// TIA Portal V18 export
DATA_BLOCK "ST10_DeviceError"   // DB1067
{ S7_Optimized_Access := 'FALSE' }
VERSION : 0.1
// stored: AutoNumber false, DBAccessibleFromOPCUA true, DBAccessibleFromWebserver true, IsOnlyStoredInLoadMemory false, IsWriteProtectedInAS false
   VAR RETAIN
      CylinderFault : Struct   // Cylinder Error（气缸错误）
         C1GoWorkFault : Bool;   // Cyl1
         C1GoHomeFault : Bool;   // Cyl1
         C1SensorPositionFault : Bool;   // Cyl1
         C1SpareFault : Bool;
         C2GoWorkFault : Bool;   // Cyl2
         C2GoHomeFault : Bool;   // Cyl2
         C2SensorPositionFault : Bool;   // Cyl2
         C2SpareFault : Bool;
         C3GoWorkFault : Bool;   // Cyl3
         C3GoHomeFault : Bool;   // Cyl3
         C3SensorPositionFault : Bool;   // Cyl3
         C3SpareFault : Bool;
         C4GoWorkFault : Bool;   // Cyl4
         C4GoHomeFault : Bool;   // Cyl4
         C4SensorPositionFault : Bool;   // Cyl4
         C4SpareFault : Bool;
         C5GoWorkFault : Bool;   // Cyl5
         C5GoHomeFault : Bool;   // Cyl5
         C5SensorPositionFault : Bool;   // Cyl5
         C5SpareFault : Bool;
         C6GoWorkFault : Bool;   // Cyl6
         C6GoHomeFault : Bool;   // Cyl6
         C6SensorPositionFault : Bool;   // Cyl6
         C6SpareFault : Bool;
         C7GoWorkFault : Bool;   // Cyl7
         C7GoHomeFault : Bool;   // Cyl7
         C7SensorPositionFault : Bool;   // Cyl7
         C7SpareFault : Bool;
         C8GoWorkFault : Bool;   // Cyl8
         C8GoHomeFault : Bool;   // Cyl8
         C8SensorPositionFault : Bool;   // Cyl8
         C8SpareFault : Bool;
         C9GoWorkFault : Bool;   // Cyl9
         C9GoHomeFault : Bool;   // Cyl9
         C9SensorPositionFault : Bool;   // Cyl9
         C9SpareFault : Bool;
         C10GoWorkFault : Bool;   // Cyl10
         C10GoHomeFault : Bool;   // Cyl10
         C10SensorPositionFault : Bool;   // Cyl10
         C10SpareFault : Bool;
         C11GoWorkFault : Bool;   // Cyl11
         C11GoHomeFault : Bool;   // Cyl11
         C11SensorPositionFault : Bool;   // Cyl11
         C11SpareFault : Bool;
         C12GoWorkFault : Bool;   // Cyl12
         C12GoHomeFault : Bool;   // Cyl12
         C12SensorPositionFault : Bool;   // Cyl12
         C12SpareFault : Bool;
         C13GoWorkFault : Bool;   // Cyl13
         C13GoHomeFault : Bool;   // Cyl13
         C13SensorPositionFault : Bool;   // Cyl13
         C13SpareFault : Bool;
         C14GoWorkFault : Bool;   // Cyl14
         C14GoHomeFault : Bool;   // Cyl14
         C14SensorPositionFault : Bool;   // Cyl14
         C14SpareFault : Bool;
         C15GoWorkFault : Bool;   // Cyl15
         C15GoHomeFault : Bool;   // Cyl15
         C15SensorPositionFault : Bool;   // Cyl15
         C15SpareFault : Bool;
         C16GoWorkFault : Bool;   // Cyl16
         C16GoHomeFault : Bool;   // Cyl16
         C16SensorPositionFault : Bool;   // Cyl16
         C16SpareFault : Bool;
         C17GoWorkFault : Bool;   // Cyl17
         C17GoHomeFault : Bool;   // Cyl17
         C17SensorPositionFault : Bool;   // Cyl17
         C17SpareFault : Bool;
         C18GoWorkFault : Bool;   // Cyl18
         C18GoHomeFault : Bool;   // Cyl18
         C18SensorPositionFault : Bool;   // Cyl18
         C18SpareFault : Bool;
         C19GoWorkFault : Bool;   // Cyl19
         C19GoHomeFault : Bool;   // Cyl19
         C19SensorPositionFault : Bool;   // Cyl19
         C19SpareFault : Bool;
         C20GoWorkFault : Bool;   // Cyl20
         C20GoHomeFault : Bool;   // Cyl20
         C20SensorPositionFault : Bool;   // Cyl20
         C20SpareFault : Bool;
         C21GoWorkFault : Bool;   // Cyl21
         C21GoHomeFault : Bool;   // Cyl21
         C21SensorPositionFault : Bool;   // Cyl21
         C21SpareFault : Bool;
         C22GoWorkFault : Bool;   // Cyl22
         C22GoHomeFault : Bool;   // Cyl22
         C22SensorPositionFault : Bool;   // Cyl22
         C22SpareFault : Bool;
         C23GoWorkFault : Bool;   // Cyl23
         C23GoHomeFault : Bool;   // Cyl23
         C23SensorPositionFault : Bool;   // Cyl23
         C23SpareFault : Bool;
         C24GoWorkFault : Bool;   // Cyl24
         C24GoHomeFault : Bool;   // Cyl24
         C24SensorPositionFault : Bool;   // Cyl24
         C24SpareFault : Bool;
         C25GoWorkFault : Bool;   // Cyl25
         C25GoHomeFault : Bool;   // Cyl25
         C25SensorPositionFault : Bool;   // Cyl25
         C25SpareFault : Bool;
         C26GoWorkFault : Bool;   // Cyl26
         C26GoHomeFault : Bool;   // Cyl26
         C26SensorPositionFault : Bool;   // Cyl26
         C26SpareFault : Bool;
         C27GoWorkFault : Bool;   // Cyl27
         C27GoHomeFault : Bool;   // Cyl27
         C27SensorPositionFault : Bool;   // Cyl27
         C27SpareFault : Bool;
         C28GoWorkFault : Bool;   // Cyl28
         C28GoHomeFault : Bool;   // Cyl28
         C28SensorPositionFault : Bool;   // Cyl28
         C28SpareFault : Bool;
         C29GoWorkFault : Bool;   // Cyl29
         C29GoHomeFault : Bool;   // Cyl29
         C29SensorPositionFault : Bool;   // Cyl29
         C29SpareFault : Bool;
         C30GoWorkFault : Bool;   // Cyl30
         C30GoHomeFault : Bool;   // Cyl30
         C30SensorPositionFault : Bool;   // Cyl30
         C30SpareFault : Bool;
         C31GoWorkFault : Bool;   // Cyl31
         C31GoHomeFault : Bool;   // Cyl31
         C31SensorPositionFault : Bool;   // Cyl31
         C31SpareFault : Bool;
         C32GoWorkFault : Bool;   // Cyl32
         C32GoHomeFault : Bool;   // Cyl32
         C32SensorPositionFault : Bool;   // Cyl32
         C32SpareFault : Bool;
         C33GoWorkFault : Bool;   // Cyl33
         C33GoHomeFault : Bool;   // Cyl33
         C33SensorPositionFault : Bool;   // Cyl33
         C33SpareFault : Bool;
         C34GoWorkFault : Bool;   // Cyl34
         C34GoHomeFault : Bool;   // Cyl34
         C34SensorPositionFault : Bool;   // Cyl34
         C34SpareFault : Bool;
         C35GoWorkFault : Bool;   // Cyl35
         C35GoHomeFault : Bool;   // Cyl35
         C35SensorPositionFault : Bool;   // Cyl35
         C35SpareFault : Bool;
         C36GoWorkFault : Bool;   // Cyl36
         C36GoHomeFault : Bool;   // Cyl36
         C36SensorPositionFault : Bool;   // Cyl36
         C36SpareFault : Bool;
         C37GoWorkFault : Bool;   // Cyl37
         C37GoHomeFault : Bool;   // Cyl37
         C37SensorPositionFault : Bool;   // Cyl37
         C37SpareFault : Bool;
         C38GoWorkFault : Bool;   // Cyl38
         C38GoHomeFault : Bool;   // Cyl38
         C38SensorPositionFault : Bool;   // Cyl38
         C38SpareFault : Bool;
         C39GoWorkFault : Bool;   // Cyl39
         C39GoHomeFault : Bool;   // Cyl39
         C39SensorPositionFault : Bool;   // Cyl39
         C39SpareFault : Bool;
         C40GoWorkFault : Bool;   // Cyl40
         C40GoHomeFault : Bool;   // Cyl40
         C40SensorPositionFault : Bool;   // Cyl40
         C40SpareFault : Bool;
         C41GoWorkFault : Bool;   // Cyl41
         C41GoHomeFault : Bool;   // Cyl41
         C41SensorPositionFault : Bool;   // Cyl41
         C41SpareFault : Bool;
         C42GoWorkFault : Bool;   // Cyl42
         C42GoHomeFault : Bool;   // Cyl42
         C42SensorPositionFault : Bool;   // Cyl42
         C42SpareFault : Bool;
         C43GoWorkFault : Bool;   // Cyl43
         C43GoHomeFault : Bool;   // Cyl43
         C43SensorPositionFault : Bool;   // Cyl43
         C43SpareFault : Bool;
         C44GoWorkFault : Bool;   // Cyl44
         C44GoHomeFault : Bool;   // Cyl44
         C44SensorPositionFault : Bool;   // Cyl44
         C44SpareFault : Bool;
         C45GoWorkFault : Bool;   // Cyl45
         C45GoHomeFault : Bool;   // Cyl45
         C45SensorPositionFault : Bool;   // Cyl45
         C45SpareFault : Bool;
         C46GoWorkFault : Bool;   // Cyl46
         C46GoHomeFault : Bool;   // Cyl46
         C46SensorPositionFault : Bool;   // Cyl46
         C46SpareFault : Bool;
         C47GoWorkFault : Bool;   // Cyl47
         C47GoHomeFault : Bool;   // Cyl47
         C47SensorPositionFault : Bool;   // Cyl47
         C47SpareFault : Bool;
         C48GoWorkFault : Bool;   // Cyl48
         C48GoHomeFault : Bool;   // Cyl48
         C48SensorPositionFault : Bool;   // Cyl48
         C48SpareFault : Bool;
         C49GoWorkFault : Bool;   // Cyl49
         C49GoHomeFault : Bool;   // Cyl49
         C49SensorPositionFault : Bool;   // Cyl49
         C49SpareFault : Bool;
         C50GoWorkFault : Bool;   // Cyl50
         C50GoHomeFault : Bool;   // Cyl50
         C50SensorPositionFault : Bool;   // Cyl50
         C50SpareFault : Bool;
         C51GoWorkFault : Bool;   // Cyl51
         C51GoHomeFault : Bool;   // Cyl51
         C51SensorPositionFault : Bool;   // Cyl51
         C51SpareFault : Bool;
         C52GoWorkFault : Bool;   // Cyl52
         C52GoHomeFault : Bool;   // Cyl52
         C52SensorPositionFault : Bool;   // Cyl52
         C52SpareFault : Bool;
         C53GoWorkFault : Bool;   // Cyl53
         C53GoHomeFault : Bool;   // Cyl53
         C53SensorPositionFault : Bool;   // Cyl53
         C53SpareFault : Bool;
         C54GoWorkFault : Bool;   // Cyl54
         C54GoHomeFault : Bool;   // Cyl54
         C54SensorPositionFault : Bool;   // Cyl54
         C54SpareFault : Bool;
         C55GoWorkFault : Bool;   // Cyl55
         C55GoHomeFault : Bool;   // Cyl55
         C55SensorPositionFault : Bool;   // Cyl55
         C55SpareFault : Bool;
         C56GoWorkFault : Bool;   // Cyl56
         C56GoHomeFault : Bool;   // Cyl56
         C56SensorPositionFault : Bool;   // Cyl56
         C56SpareFault : Bool;
         C57GoWorkFault : Bool;   // Cyl57
         C57GoHomeFault : Bool;   // Cyl57
         C57SensorPositionFault : Bool;   // Cyl57
         C57SpareFault : Bool;
         C58GoWorkFault : Bool;   // Cyl58
         C58GoHomeFault : Bool;   // Cyl58
         C58SensorPositionFault : Bool;   // Cyl58
         C58SpareFault : Bool;
         C59GoWorkFault : Bool;   // Cyl59
         C59GoHomeFault : Bool;   // Cyl59
         C59SensorPositionFault : Bool;   // Cyl59
         C59SpareFault : Bool;
         C60GoWorkFault : Bool;   // Cyl60
         C60GoHomeFault : Bool;   // Cyl60
         C60SensorPositionFault : Bool;   // Cyl60
         C60SpareFault : Bool;
         C61GoWorkFault : Bool;   // Cyl61
         C61GoHomeFault : Bool;   // Cyl61
         C61SensorPositionFault : Bool;   // Cyl61
         C61SpareFault : Bool;
         C62GoWorkFault : Bool;   // Cyl62
         C62GoHomeFault : Bool;   // Cyl62
         C62SensorPositionFault : Bool;   // Cyl62
         C62SpareFault : Bool;
         C63GoWorkFault : Bool;   // Cyl63
         C63GoHomeFault : Bool;   // Cyl63
         C63SensorPositionFault : Bool;   // Cyl63
         C63SpareFault : Bool;
         C64GoWorkFault : Bool;   // Cyl64
         C64GoHomeFault : Bool;   // Cyl64
         C64SensorPositionFault : Bool;   // Cyl64
         C64SpareFault : Bool;
         C65GoWorkFault : Bool;   // Cyl65
         C65GoHomeFault : Bool;   // Cyl65
         C65SensorPositionFault : Bool;   // Cyl65
         C65SpareFault : Bool;
         C66GoWorkFault : Bool;   // Cyl66
         C66GoHomeFault : Bool;   // Cyl66
         C66SensorPositionFault : Bool;   // Cyl66
         C66SpareFault : Bool;
         C67GoWorkFault : Bool;   // Cyl67
         C67GoHomeFault : Bool;   // Cyl67
         C67SensorPositionFault : Bool;   // Cyl67
         C67SpareFault : Bool;
         C68GoWorkFault : Bool;   // Cyl68
         C68GoHomeFault : Bool;   // Cyl68
         C68SensorPositionFault : Bool;   // Cyl68
         C68SpareFault : Bool;
         C69GoWorkFault : Bool;   // Cyl69
         C69GoHomeFault : Bool;   // Cyl69
         C69SensorPositionFault : Bool;   // Cyl69
         C69SpareFault : Bool;
         C70GoWorkFault : Bool;   // Cyl70
         C70GoHomeFault : Bool;   // Cyl70
         C70SensorPositionFault : Bool;   // Cyl70
         C70SpareFault : Bool;
         C71GoWorkFault : Bool;   // Cyl71
         C71GoHomeFault : Bool;   // Cyl71
         C71SensorPositionFault : Bool;   // Cyl71
         C71SpareFault : Bool;
         C72GoWorkFault : Bool;   // Cyl72
         C72GoHomeFault : Bool;   // Cyl72
         C72SensorPositionFault : Bool;   // Cyl72
         C72SpareFault : Bool;
         C73GoWorkFault : Bool;   // Cyl73
         C73GoHomeFault : Bool;   // Cyl73
         C73SensorPositionFault : Bool;   // Cyl73
         C73SpareFault : Bool;
         C74GoWorkFault : Bool;   // Cyl74
         C74GoHomeFault : Bool;   // Cyl74
         C74SensorPositionFault : Bool;   // Cyl74
         C74SpareFault : Bool;
         C75GoWorkFault : Bool;   // Cyl75
         C75GoHomeFault : Bool;   // Cyl75
         C75SensorPositionFault : Bool;   // Cyl75
         C75SpareFault : Bool;
         C76GoWorkFault : Bool;   // Cyl76
         C76GoHomeFault : Bool;   // Cyl76
         C76SensorPositionFault : Bool;   // Cyl76
         C76SpareFault : Bool;
         C77GoWorkFault : Bool;   // Cyl77
         C77GoHomeFault : Bool;   // Cyl77
         C77SensorPositionFault : Bool;   // Cyl77
         C77SpareFault : Bool;
         C78GoWorkFault : Bool;   // Cyl78
         C78GoHomeFault : Bool;   // Cyl78
         C78SensorPositionFault : Bool;   // Cyl78
         C78SpareFault : Bool;
         C79GoWorkFault : Bool;   // Cyl79
         C79GoHomeFault : Bool;   // Cyl79
         C79SensorPositionFault : Bool;   // Cyl79
         C79SpareFault : Bool;
         C80GoWorkFault : Bool;   // Cyl80
         C80GoHomeFault : Bool;   // Cyl80
         C80SensorPositionFault : Bool;   // Cyl80
         C80SpareFault : Bool;
         C81GoWorkFault : Bool;   // Cyl81
         C81GoHomeFault : Bool;   // Cyl81
         C81SensorPositionFault : Bool;   // Cyl81
         C81SpareFault : Bool;
         C82GoWorkFault : Bool;   // Cyl82
         C82GoHomeFault : Bool;   // Cyl82
         C82SensorPositionFault : Bool;   // Cyl82
         C82SpareFault : Bool;
         C83GoWorkFault : Bool;   // Cyl83
         C83GoHomeFault : Bool;   // Cyl83
         C83SensorPositionFault : Bool;   // Cyl83
         C83SpareFault : Bool;
         C84GoWorkFault : Bool;   // Cyl84
         C84GoHomeFault : Bool;   // Cyl84
         C84SensorPositionFault : Bool;   // Cyl84
         C84SpareFault : Bool;
         C85GoWorkFault : Bool;   // Cyl85
         C85GoHomeFault : Bool;   // Cyl85
         C85SensorPositionFault : Bool;   // Cyl85
         C85SpareFault : Bool;
         C86GoWorkFault : Bool;   // Cyl86
         C86GoHomeFault : Bool;   // Cyl86
         C86SensorPositionFault : Bool;   // Cyl86
         C86SpareFault : Bool;
         C87GoWorkFault : Bool;   // Cyl87
         C87GoHomeFault : Bool;   // Cyl87
         C87SensorPositionFault : Bool;   // Cyl87
         C87SpareFault : Bool;
         C88GoWorkFault : Bool;   // Cyl88
         C88GoHomeFault : Bool;   // Cyl88
         C88SensorPositionFault : Bool;   // Cyl88
         C88SpareFault : Bool;
         C89GoWorkFault : Bool;   // Cyl89
         C89GoHomeFault : Bool;   // Cyl89
         C89SensorPositionFault : Bool;   // Cyl89
         C89SpareFault : Bool;
         C90GoWorkFault : Bool;   // Cyl90
         C90GoHomeFault : Bool;   // Cyl90
         C90SensorPositionFault : Bool;   // Cyl90
         C90SpareFault : Bool;
         C91GoWorkFault : Bool;   // Cyl91
         C91GoHomeFault : Bool;   // Cyl91
         C91SensorPositionFault : Bool;   // Cyl91
         C91SpareFault : Bool;
         C92GoWorkFault : Bool;   // Cyl92
         C92GoHomeFault : Bool;   // Cyl92
         C92SensorPositionFault : Bool;   // Cyl92
         C92SpareFault : Bool;
         C93GoWorkFault : Bool;   // Cyl93
         C93GoHomeFault : Bool;   // Cyl93
         C93SensorPositionFault : Bool;   // Cyl93
         C93SpareFault : Bool;
         C94GoWorkFault : Bool;   // Cyl94
         C94GoHomeFault : Bool;   // Cyl94
         C94SensorPositionFault : Bool;   // Cyl94
         C94SpareFault : Bool;
         C95GoWorkFault : Bool;   // Cyl95
         C95GoHomeFault : Bool;   // Cyl95
         C95SensorPositionFault : Bool;   // Cyl95
         C95SpareFault : Bool;
         C96GoWorkFault : Bool;   // Cyl96
         C96GoHomeFault : Bool;   // Cyl96
         C96SensorPositionFault : Bool;   // Cyl96
         C96SpareFault : Bool;
         C97GoWorkFault : Bool;   // Cyl97
         C97GoHomeFault : Bool;   // Cyl97
         C97SensorPositionFault : Bool;   // Cyl97
         C97SpareFault : Bool;
         C98GoWorkFault : Bool;   // Cyl98
         C98GoHomeFault : Bool;   // Cyl98
         C98SensorPositionFault : Bool;   // Cyl98
         C98SpareFault : Bool;
         C99GoWorkFault : Bool;   // Cyl99
         C99GoHomeFault : Bool;   // Cyl99
         C99SensorPositionFault : Bool;   // Cyl99
         C99SpareFault : Bool;
         C100GoWorkFault : Bool;   // Cyl100
         C100GoHomeFault : Bool;   // Cyl100
         C100SensorPositionFault : Bool;   // Cyl100
         C100SpareFault : Bool;
         C101GoWorkFault : Bool;   // Cyl101
         C101GoHomeFault : Bool;   // Cyl101
         C101SensorPositionFault : Bool;   // Cyl101
         C101SpareFault : Bool;
         C102GoWorkFault : Bool;   // Cyl102
         C102GoHomeFault : Bool;   // Cyl102
         C102SensorPositionFault : Bool;   // Cyl102
         C102SpareFault : Bool;
         C103GoWorkFault : Bool;   // Cyl103
         C103GoHomeFault : Bool;   // Cyl103
         C103SensorPositionFault : Bool;   // Cyl103
         C103SpareFault : Bool;
         C104GoWorkFault : Bool;   // Cyl104
         C104GoHomeFault : Bool;   // Cyl104
         C104SensorPositionFault : Bool;   // Cyl104
         C104SpareFault : Bool;
         C105GoWorkFault : Bool;   // Cyl105
         C105GoHomeFault : Bool;   // Cyl105
         C105SensorPositionFault : Bool;   // Cyl105
         C105SpareFault : Bool;
         C106GoWorkFault : Bool;   // Cyl106
         C106GoHomeFault : Bool;   // Cyl106
         C106SensorPositionFault : Bool;   // Cyl106
         C106SpareFault : Bool;
         C107GoWorkFault : Bool;   // Cyl107
         C107GoHomeFault : Bool;   // Cyl107
         C107SensorPositionFault : Bool;   // Cyl107
         C107SpareFault : Bool;
         C108GoWorkFault : Bool;   // Cyl108
         C108GoHomeFault : Bool;   // Cyl108
         C108SensorPositionFault : Bool;   // Cyl108
         C108SpareFault : Bool;
         C109GoWorkFault : Bool;   // Cyl109
         C109GoHomeFault : Bool;   // Cyl109
         C109SensorPositionFault : Bool;   // Cyl109
         C109SpareFault : Bool;
         C110GoWorkFault : Bool;   // Cyl110
         C110GoHomeFault : Bool;   // Cyl110
         C110SensorPositionFault : Bool;   // Cyl110
         C110SpareFault : Bool;
         C111GoWorkFault : Bool;   // Cyl111
         C111GoHomeFault : Bool;   // Cyl111
         C111SensorPositionFault : Bool;   // Cyl111
         C111SpareFault : Bool;
         C112GoWorkFault : Bool;   // Cyl112
         C112GoHomeFault : Bool;   // Cyl112
         C112SensorPositionFault : Bool;   // Cyl112
         C112SpareFault : Bool;
         C113GoWorkFault : Bool;   // Cyl113
         C113GoHomeFault : Bool;   // Cyl113
         C113SensorPositionFault : Bool;   // Cyl113
         C113SpareFault : Bool;
         C114GoWorkFault : Bool;   // Cyl114
         C114GoHomeFault : Bool;   // Cyl114
         C114SensorPositionFault : Bool;   // Cyl114
         C114SpareFault : Bool;
         C115GoWorkFault : Bool;   // Cyl115
         C115GoHomeFault : Bool;   // Cyl115
         C115SensorPositionFault : Bool;   // Cyl115
         C115SpareFault : Bool;
         C116GoWorkFault : Bool;   // Cyl116
         C116GoHomeFault : Bool;   // Cyl116
         C116SensorPositionFault : Bool;   // Cyl116
         C116SpareFault : Bool;
         C117GoWorkFault : Bool;   // Cyl117
         C117GoHomeFault : Bool;   // Cyl117
         C117SensorPositionFault : Bool;   // Cyl117
         C117SpareFault : Bool;
         C118GoWorkFault : Bool;   // Cyl118
         C118GoHomeFault : Bool;   // Cyl118
         C118SensorPositionFault : Bool;   // Cyl118
         C118SpareFault : Bool;
         C119GoWorkFault : Bool;   // Cyl119
         C119GoHomeFault : Bool;   // Cyl119
         C119SensorPositionFault : Bool;   // Cyl119
         C119SpareFault : Bool;
         C120GoWorkFault : Bool;   // Cyl120
         C120GoHomeFault : Bool;   // Cyl120
         C120SensorPositionFault : Bool;   // Cyl120
         C120SpareFault : Bool;
         C121GoWorkFault : Bool;   // Cyl121
         C121GoHomeFault : Bool;   // Cyl121
         C121SensorPositionFault : Bool;   // Cyl121
         C121SpareFault : Bool;
         C122GoWorkFault : Bool;   // Cyl122
         C122GoHomeFault : Bool;   // Cyl122
         C122SensorPositionFault : Bool;   // Cyl122
         C122SpareFault : Bool;
         C123GoWorkFault : Bool;   // Cyl123
         C123GoHomeFault : Bool;   // Cyl123
         C123SensorPositionFault : Bool;   // Cyl123
         C123SpareFault : Bool;
         C124GoWorkFault : Bool;   // Cyl124
         C124GoHomeFault : Bool;   // Cyl124
         C124SensorPositionFault : Bool;   // Cyl124
         C124SpareFault : Bool;
         C125GoWorkFault : Bool;   // Cyl125
         C125GoHomeFault : Bool;   // Cyl125
         C125SensorPositionFault : Bool;   // Cyl125
         C125SpareFault : Bool;
         C126GoWorkFault : Bool;   // Cyl126
         C126GoHomeFault : Bool;   // Cyl126
         C126SensorPositionFault : Bool;   // Cyl126
         C126SpareFault : Bool;
         C127GoWorkFault : Bool;   // Cyl127
         C127GoHomeFault : Bool;   // Cyl127
         C127SensorPositionFault : Bool;   // Cyl127
         C127SpareFault : Bool;
         C128GoWorkFault : Bool;   // Cyl128
         C128GoHomeFault : Bool;   // Cyl128
         C128SensorPositionFault : Bool;   // Cyl128
         C128SpareFault : Bool;
         C129GoWorkFault : Bool;   // Cyl129
         C129GoHomeFault : Bool;   // Cyl129
         C129SensorPositionFault : Bool;   // Cyl129
         C129SpareFault : Bool;
         C130GoWorkFault : Bool;   // Cyl130
         C130GoHomeFault : Bool;   // Cyl130
         C130SensorPositionFault : Bool;   // Cyl130
         C130SpareFault : Bool;
         C131GoWorkFault : Bool;   // Cyl131
         C131GoHomeFault : Bool;   // Cyl131
         C131SensorPositionFault : Bool;   // Cyl131
         C131SpareFault : Bool;
         C132GoWorkFault : Bool;   // Cyl132
         C132GoHomeFault : Bool;   // Cyl132
         C132SensorPositionFault : Bool;   // Cyl132
         C132SpareFault : Bool;
         C133GoWorkFault : Bool;   // Cyl133
         C133GoHomeFault : Bool;   // Cyl133
         C133SensorPositionFault : Bool;   // Cyl133
         C133SpareFault : Bool;
         C134GoWorkFault : Bool;   // Cyl134
         C134GoHomeFault : Bool;   // Cyl134
         C134SensorPositionFault : Bool;   // Cyl134
         C134SpareFault : Bool;
         C135GoWorkFault : Bool;   // Cyl135
         C135GoHomeFault : Bool;   // Cyl135
         C135SensorPositionFault : Bool;   // Cyl135
         C135SpareFault : Bool;
         C136GoWorkFault : Bool;   // Cyl136
         C136GoHomeFault : Bool;   // Cyl136
         C136SensorPositionFault : Bool;   // Cyl136
         C136SpareFault : Bool;
         C137GoWorkFault : Bool;   // Cyl137
         C137GoHomeFault : Bool;   // Cyl137
         C137SensorPositionFault : Bool;   // Cyl137
         C137SpareFault : Bool;
         C138GoWorkFault : Bool;   // Cyl138
         C138GoHomeFault : Bool;   // Cyl138
         C138SensorPositionFault : Bool;   // Cyl138
         C138SpareFault : Bool;
         C139GoWorkFault : Bool;   // Cyl139
         C139GoHomeFault : Bool;   // Cyl139
         C139SensorPositionFault : Bool;   // Cyl139
         C139SpareFault : Bool;
         C140GoWorkFault : Bool;   // Cyl140
         C140GoHomeFault : Bool;   // Cyl140
         C140SensorPositionFault : Bool;   // Cyl140
         C140SpareFault : Bool;
         C141GoWorkFault : Bool;   // Cyl141
         C141GoHomeFault : Bool;   // Cyl141
         C141SensorPositionFault : Bool;   // Cyl141
         C141SpareFault : Bool;
         C142GoWorkFault : Bool;   // Cyl142
         C142GoHomeFault : Bool;   // Cyl142
         C142SensorPositionFault : Bool;   // Cyl142
         C142SpareFault : Bool;
         C143GoWorkFault : Bool;   // Cyl143
         C143GoHomeFault : Bool;   // Cyl143
         C143SensorPositionFault : Bool;   // Cyl143
         C143SpareFault : Bool;
         C144GoWorkFault : Bool;   // Cyl144
         C144GoHomeFault : Bool;   // Cyl144
         C144SensorPositionFault : Bool;   // Cyl144
         C144SpareFault : Bool;
         C145GoWorkFault : Bool;   // Cyl145
         C145GoHomeFault : Bool;   // Cyl145
         C145SensorPositionFault : Bool;   // Cyl145
         C145SpareFault : Bool;
         C146GoWorkFault : Bool;   // Cyl146
         C146GoHomeFault : Bool;   // Cyl146
         C146SensorPositionFault : Bool;   // Cyl146
         C146SpareFault : Bool;
         C147GoWorkFault : Bool;   // Cyl147
         C147GoHomeFault : Bool;   // Cyl147
         C147SensorPositionFault : Bool;   // Cyl147
         C147SpareFault : Bool;
         C148GoWorkFault : Bool;   // Cyl148
         C148GoHomeFault : Bool;   // Cyl148
         C148SensorPositionFault : Bool;   // Cyl148
         C148SpareFault : Bool;
         C149GoWorkFault : Bool;   // Cyl149
         C149GoHomeFault : Bool;   // Cyl149
         C149SensorPositionFault : Bool;   // Cyl149
         C149SpareFault : Bool;
         C150GoWorkFault : Bool;   // Cyl150
         C150GoHomeFault : Bool;   // Cyl150
         C150SensorPositionFault : Bool;   // Cyl150
         C150SpareFault : Bool;
         C151GoWorkFault : Bool;   // Cyl151
         C151GoHomeFault : Bool;   // Cyl151
         C151SensorPositionFault : Bool;   // Cyl151
         C151SpareFault : Bool;
         C152GoWorkFault : Bool;   // Cyl152
         C152GoHomeFault : Bool;   // Cyl152
         C152SensorPositionFault : Bool;   // Cyl152
         C152SpareFault : Bool;
         C153GoWorkFault : Bool;   // Cyl153
         C153GoHomeFault : Bool;   // Cyl153
         C153SensorPositionFault : Bool;   // Cyl153
         C153SpareFault : Bool;
         C154GoWorkFault : Bool;   // Cyl154
         C154GoHomeFault : Bool;   // Cyl154
         C154SensorPositionFault : Bool;   // Cyl154
         C154SpareFault : Bool;
         C155GoWorkFault : Bool;   // Cyl155
         C155GoHomeFault : Bool;   // Cyl155
         C155SensorPositionFault : Bool;   // Cyl155
         C155SpareFault : Bool;
         C156GoWorkFault : Bool;   // Cyl156
         C156GoHomeFault : Bool;   // Cyl156
         C156SensorPositionFault : Bool;   // Cyl156
         C156SpareFault : Bool;
         C157GoWorkFault : Bool;   // Cyl157
         C157GoHomeFault : Bool;   // Cyl157
         C157SensorPositionFault : Bool;   // Cyl157
         C157SpareFault : Bool;
         C158GoWorkFault : Bool;   // Cyl158
         C158GoHomeFault : Bool;   // Cyl158
         C158SensorPositionFault : Bool;   // Cyl158
         C158SpareFault : Bool;
         C159GoWorkFault : Bool;   // Cyl159
         C159GoHomeFault : Bool;   // Cyl159
         C159SensorPositionFault : Bool;   // Cyl159
         C159SpareFault : Bool;
         C160GoWorkFault : Bool;   // Cyl160
         C160GoHomeFault : Bool;   // Cyl160
         C160SensorPositionFault : Bool;   // Cyl160
         C160SpareFault : Bool;
         C161GoWorkFault : Bool;   // Cyl161
         C161GoHomeFault : Bool;   // Cyl161
         C161SensorPositionFault : Bool;   // Cyl161
         C161SpareFault : Bool;
         C162GoWorkFault : Bool;   // Cyl162
         C162GoHomeFault : Bool;   // Cyl162
         C162SensorPositionFault : Bool;   // Cyl162
         C162SpareFault : Bool;
         C163GoWorkFault : Bool;   // Cyl163
         C163GoHomeFault : Bool;   // Cyl163
         C163SensorPositionFault : Bool;   // Cyl163
         C163SpareFault : Bool;
         C164GoWorkFault : Bool;   // Cyl164
         C164GoHomeFault : Bool;   // Cyl164
         C164SensorPositionFault : Bool;   // Cyl164
         C164SpareFault : Bool;
         C165GoWorkFault : Bool;   // Cyl165
         C165GoHomeFault : Bool;   // Cyl165
         C165SensorPositionFault : Bool;   // Cyl165
         C165SpareFault : Bool;
         C166GoWorkFault : Bool;   // Cyl166
         C166GoHomeFault : Bool;   // Cyl166
         C166SensorPositionFault : Bool;   // Cyl166
         C166SpareFault : Bool;
         C167GoWorkFault : Bool;   // Cyl167
         C167GoHomeFault : Bool;   // Cyl167
         C167SensorPositionFault : Bool;   // Cyl167
         C167SpareFault : Bool;
         C168GoWorkFault : Bool;   // Cyl168
         C168GoHomeFault : Bool;   // Cyl168
         C168SensorPositionFault : Bool;   // Cyl168
         C168SpareFault : Bool;
         C169GoWorkFault : Bool;   // Cyl169
         C169GoHomeFault : Bool;   // Cyl169
         C169SensorPositionFault : Bool;   // Cyl169
         C169SpareFault : Bool;
         C170GoWorkFault : Bool;   // Cyl170
         C170GoHomeFault : Bool;   // Cyl170
         C170SensorPositionFault : Bool;   // Cyl170
         C170SpareFault : Bool;
         C171GoWorkFault : Bool;   // Cyl171
         C171GoHomeFault : Bool;   // Cyl171
         C171SensorPositionFault : Bool;   // Cyl171
         C171SpareFault : Bool;
         C172GoWorkFault : Bool;   // Cyl172
         C172GoHomeFault : Bool;   // Cyl172
         C172SensorPositionFault : Bool;   // Cyl172
         C172SpareFault : Bool;
         C173GoWorkFault : Bool;   // Cyl173
         C173GoHomeFault : Bool;   // Cyl173
         C173SensorPositionFault : Bool;   // Cyl173
         C173SpareFault : Bool;
         C174GoWorkFault : Bool;   // Cyl174
         C174GoHomeFault : Bool;   // Cyl174
         C174SensorPositionFault : Bool;   // Cyl174
         C174SpareFault : Bool;
         C175GoWorkFault : Bool;   // Cyl175
         C175GoHomeFault : Bool;   // Cyl175
         C175SensorPositionFault : Bool;   // Cyl175
         C175SpareFault : Bool;
         C176GoWorkFault : Bool;   // Cyl176
         C176GoHomeFault : Bool;   // Cyl176
         C176SensorPositionFault : Bool;   // Cyl176
         C176SpareFault : Bool;
         C177GoWorkFault : Bool;   // Cyl177
         C177GoHomeFault : Bool;   // Cyl177
         C177SensorPositionFault : Bool;   // Cyl177
         C177SpareFault : Bool;
         C178GoWorkFault : Bool;   // Cyl178
         C178GoHomeFault : Bool;   // Cyl178
         C178SensorPositionFault : Bool;   // Cyl178
         C178SpareFault : Bool;
         C179GoWorkFault : Bool;   // Cyl179
         C179GoHomeFault : Bool;   // Cyl179
         C179SensorPositionFault : Bool;   // Cyl179
         C179SpareFault : Bool;
         C180GoWorkFault : Bool;   // Cyl180
         C180GoHomeFault : Bool;   // Cyl180
         C180SensorPositionFault : Bool;   // Cyl180
         C180SpareFault : Bool;
         C181GoWorkFault : Bool;   // Cyl181
         C181GoHomeFault : Bool;   // Cyl181
         C181SensorPositionFault : Bool;   // Cyl181
         C181SpareFault : Bool;
         C182GoWorkFault : Bool;   // Cyl182
         C182GoHomeFault : Bool;   // Cyl182
         C182SensorPositionFault : Bool;   // Cyl182
         C182SpareFault : Bool;
         C183GoWorkFault : Bool;   // Cyl183
         C183GoHomeFault : Bool;   // Cyl183
         C183SensorPositionFault : Bool;   // Cyl183
         C183SpareFault : Bool;
         C184GoWorkFault : Bool;   // Cyl184
         C184GoHomeFault : Bool;   // Cyl184
         C184SensorPositionFault : Bool;   // Cyl184
         C184SpareFault : Bool;
         C185GoWorkFault : Bool;   // Cyl185
         C185GoHomeFault : Bool;   // Cyl185
         C185SensorPositionFault : Bool;   // Cyl185
         C185SpareFault : Bool;
         C186GoWorkFault : Bool;   // Cyl186
         C186GoHomeFault : Bool;   // Cyl186
         C186SensorPositionFault : Bool;   // Cyl186
         C186SpareFault : Bool;
         C187GoWorkFault : Bool;   // Cyl187
         C187GoHomeFault : Bool;   // Cyl187
         C187SensorPositionFault : Bool;   // Cyl187
         C187SpareFault : Bool;
         C188GoWorkFault : Bool;   // Cyl188
         C188GoHomeFault : Bool;   // Cyl188
         C188SensorPositionFault : Bool;   // Cyl188
         C188SpareFault : Bool;
         C189GoWorkFault : Bool;   // Cyl189
         C189GoHomeFault : Bool;   // Cyl189
         C189SensorPositionFault : Bool;   // Cyl189
         C189SpareFault : Bool;
         C190GoWorkFault : Bool;   // Cyl190
         C190GoHomeFault : Bool;   // Cyl190
         C190SensorPositionFault : Bool;   // Cyl190
         C190SpareFault : Bool;
         C191GoWorkFault : Bool;   // Cyl191
         C191GoHomeFault : Bool;   // Cyl191
         C191SensorPositionFault : Bool;   // Cyl191
         C191SpareFault : Bool;
         C192GoWorkFault : Bool;   // Cyl192
         C192GoHomeFault : Bool;   // Cyl192
         C192SensorPositionFault : Bool;   // Cyl192
         C192SpareFault : Bool;
         C193GoWorkFault : Bool;   // Cyl193
         C193GoHomeFault : Bool;   // Cyl193
         C193SensorPositionFault : Bool;   // Cyl193
         C193SpareFault : Bool;
         C194GoWorkFault : Bool;   // Cyl194
         C194GoHomeFault : Bool;   // Cyl194
         C194SensorPositionFault : Bool;   // Cyl194
         C194SpareFault : Bool;
         C195GoWorkFault : Bool;   // Cyl195
         C195GoHomeFault : Bool;   // Cyl195
         C195SensorPositionFault : Bool;   // Cyl195
         C195SpareFault : Bool;
         C196GoWorkFault : Bool;   // Cyl196
         C196GoHomeFault : Bool;   // Cyl196
         C196SensorPositionFault : Bool;   // Cyl196
         C196SpareFault : Bool;
         C197GoWorkFault : Bool;   // Cyl197
         C197GoHomeFault : Bool;   // Cyl197
         C197SensorPositionFault : Bool;   // Cyl197
         C197SpareFault : Bool;
         C198GoWorkFault : Bool;   // Cyl198
         C198GoHomeFault : Bool;   // Cyl198
         C198SensorPositionFault : Bool;   // Cyl198
         C198SpareFault : Bool;
         C199GoWorkFault : Bool;   // Cyl199
         C199GoHomeFault : Bool;   // Cyl199
         C199SensorPositionFault : Bool;   // Cyl199
         C199SpareFault : Bool;
         C200GoWorkFault : Bool;   // Cyl200
         C200GoHomeFault : Bool;   // Cyl200
         C200SensorPositionFault : Bool;   // Cyl200
         C200SpareFault : Bool;
      END_STRUCT;
      "A" : Struct   // D-提升机顶升入口电机1错误
         A1TableScan : Struct   // Conveyor motor Breaker tripped,please check input Ix.x
            LightCuritTouch : Bool;
            ScanCodeNG : Bool;
            "3" : Bool;
            "4" : Bool;
            "5" : Bool;
            "6" : Bool;
            "7" : Bool;
            "8" : Bool;
            "9" : Bool;
            "10" : Bool;
            "11" : Bool;
            "12" : Bool;
            "13" : Bool;
            "14" : Bool;
            "15" : Bool;
            "16" : Bool;
         END_STRUCT;
         A1TableUnloading : Struct   // Conveyor motor start abnormal,please check output Qx.x
            LackMaterial : Bool;
            RingCheckExist : Bool;
            "3" : Bool;
            "4" : Bool;
            "5" : Bool;
            "6" : Bool;
            "7" : Bool;
            "8" : Bool;
            "9" : Bool;
            "10" : Bool;
            "11" : Bool;
            "12" : Bool;
            "13" : Bool;
            "14" : Bool;
            "15" : Bool;
            "16" : Bool;
         END_STRUCT;
         A1RotaryScan : Struct
            ProductAnomaly : Bool;
            PartMissing : Bool;
            "3" : Bool;
            "4" : Bool;
            "5" : Bool;
            "6" : Bool;
            "7" : Bool;
            "8" : Bool;
            "9" : Bool;
            "10" : Bool;
            "11" : Bool;
            "12" : Bool;
            "13" : Bool;
            "14" : Bool;
            "15" : Bool;
            "16" : Bool;
         END_STRUCT;
         A1FixtureCodeScan : Struct
            ReadNG_1 : Bool;
            ReadNG_2 : Bool;
            ReadNG_3 : Bool;
            ReadNG_4 : Bool;
            ReadNG_5 : Bool;
            ReadNG_6 : Bool;
            ReadNG_7 : Bool;
            ReadNG_8 : Bool;
            ReadNG_9 : Bool;
            ReadNG_10 : Bool;
            ReadNG_11 : Bool;
            ReadNG_12 : Bool;
            ReadNG_13 : Bool;
            "14" : Bool;
            "15" : Bool;
            "16" : Bool;
         END_STRUCT;
         A2TableScan : Struct
            LightCuritTouch : Bool;
            ScanCodeNG : Bool;
            "3" : Bool;
            "4" : Bool;
            "5" : Bool;
            "6" : Bool;
            "7" : Bool;
            "8" : Bool;
            "9" : Bool;
            "10" : Bool;
            "11" : Bool;
            "12" : Bool;
            "13" : Bool;
            "14" : Bool;
            "15" : Bool;
            "16" : Bool;
         END_STRUCT;
         A2TableUnloading : Struct
            LackMaterial : Bool;
            RingCheckExist : Bool;
            "3" : Bool;
            "4" : Bool;
            "5" : Bool;
            "6" : Bool;
            "7" : Bool;
            "8" : Bool;
            "9" : Bool;
            "10" : Bool;
            "11" : Bool;
            "12" : Bool;
            "13" : Bool;
            "14" : Bool;
            "15" : Bool;
            "16" : Bool;
         END_STRUCT;
         A2RotaryScan : Struct
            "1" : Bool;
            "2" : Bool;
            "3" : Bool;
            "4" : Bool;
            "5" : Bool;
            "6" : Bool;
            "7" : Bool;
            "8" : Bool;
            "9" : Bool;
            "10" : Bool;
            "11" : Bool;
            "12" : Bool;
            "13" : Bool;
            "14" : Bool;
            "15" : Bool;
            "16" : Bool;
         END_STRUCT;
         A2FixtureCodeScan : Struct
            ReadNG_1 : Bool;
            ReadNG_2 : Bool;
            ReadNG_3 : Bool;
            ReadNG_4 : Bool;
            ReadNG_5 : Bool;
            ReadNG_6 : Bool;
            ReadNG_7 : Bool;
            ReadNG_8 : Bool;
            ReadNG_9 : Bool;
            ReadNG_10 : Bool;
            ReadNG_11 : Bool;
            ReadNG_12 : Bool;
            ReadNG_13 : Bool;
            "14" : Bool;
            "15" : Bool;
            "16" : Bool;
         END_STRUCT;
         Other : Struct
            Servo_380A1 : Bool;
            Servo_381A1 : Bool;
            Servo_383A1 : Bool;
            "4" : Bool;
            "5" : Bool;
            "6" : Bool;
            "7" : Bool;
            "8" : Bool;
            "9" : Bool;
            "10" : Bool;
            "11" : Bool;
            "12" : Bool;
            "13" : Bool;
            "14" : Bool;
            "15" : Bool;
            "16" : Bool;
         END_STRUCT;
         A_Spare_2 : Struct
            Servo_380A1 : Bool;
            Servo_381A1 : Bool;
            Scan_800A1 : Bool;
            Scan_801A1 : Bool;
            Scan_804A1 : Bool;
            "6" : Bool;
            "7" : Bool;
            "8" : Bool;
            "9" : Bool;
            "10" : Bool;
            "11" : Bool;
            "12" : Bool;
            "13" : Bool;
            "14" : Bool;
            "15" : Bool;
            "16" : Bool;
         END_STRUCT;
      END_STRUCT;
      "B" : Struct   // D-提升机顶升出口电机1错误
         B1Press : Struct   // Conveyor motor Breaker tripped,please check input Ix.x
            StatusError : Bool;
            ShaftSensorCheckError : Bool;
            RingSensorCheckError : Bool;
            "4" : Bool;
            "5" : Bool;
            "6" : Bool;
            "7" : Bool;
            "8" : Bool;
            "9" : Bool;
            "10" : Bool;
            "11" : Bool;
            "12" : Bool;
            "13" : Bool;
            "14" : Bool;
            "15" : Bool;
            "16" : Bool;
         END_STRUCT;
         B2Press : Struct   // Conveyor motor start abnormal,please check output Qx.x
            StatusError : Bool;
            ShaftSensorCheckError : Bool;
            RingSensorCheckError : Bool;
            "4" : Bool;
            "5" : Bool;
            "6" : Bool;
            "7" : Bool;
            "8" : Bool;
            "9" : Bool;
            "10" : Bool;
            "11" : Bool;
            "12" : Bool;
            "13" : Bool;
            "14" : Bool;
            "15" : Bool;
            "16" : Bool;
         END_STRUCT;
         B_Spare_1 : Struct
            Kistler_Press1_372A1 : Bool;
            Scan_806A1 : Bool;
            Kistler_Press2_375A1 : Bool;
            "4" : Bool;
            "5" : Bool;
            "6" : Bool;
            "7" : Bool;
            "8" : Bool;
            "9" : Bool;
            "10" : Bool;
            "11" : Bool;
            "12" : Bool;
            "13" : Bool;
            "14" : Bool;
            "15" : Bool;
            "16" : Bool;
         END_STRUCT;
         B_Spare_2 : Struct
            "1" : Bool;
            "2" : Bool;
            "3" : Bool;
            "4" : Bool;
            "5" : Bool;
            "6" : Bool;
            "7" : Bool;
            "8" : Bool;
            "9" : Bool;
            "10" : Bool;
            "11" : Bool;
            "12" : Bool;
            "13" : Bool;
            "14" : Bool;
            "15" : Bool;
            "16" : Bool;
         END_STRUCT;
         B_Spare_3 : Struct
            "1" : Bool;
            "2" : Bool;
            "3" : Bool;
            "4" : Bool;
            "5" : Bool;
            "6" : Bool;
            "7" : Bool;
            "8" : Bool;
            "9" : Bool;
            "10" : Bool;
            "11" : Bool;
            "12" : Bool;
            "13" : Bool;
            "14" : Bool;
            "15" : Bool;
            "16" : Bool;
         END_STRUCT;
      END_STRUCT;
      C : Struct   // E-线体线体电机1错误
         CGlueing : Struct   // Conveyor motor Breaker tripped,please check input Ix.x
            SysError : Bool;
            StatusError : Bool;
            Servo_383A1 : Bool;
            Z : Bool;
            X : Bool;
            Y : Bool;
            "7" : Bool;
            "8" : Bool;
            "9" : Bool;
            "10" : Bool;
            "11" : Bool;
            "12" : Bool;
            "13" : Bool;
            "14" : Bool;
            "15" : Bool;
            "16" : Bool;
         END_STRUCT;
         Other : Struct
            Servo_383A1 : Bool;
            Z : Bool;
            X : Bool;
            Y : Bool;
            "5" : Bool;
            "6" : Bool;
            "7" : Bool;
            "8" : Bool;
            "9" : Bool;
            "10" : Bool;
            "11" : Bool;
            "12" : Bool;
            "13" : Bool;
            "14" : Bool;
            "15" : Bool;
            "16" : Bool;
         END_STRUCT;
         C_Spare_2 : Struct
            Servo_382A1 : Bool;
            IV3_810A1 : Bool;
            IV3_811A1 : Bool;
            GluingDeviceReady : Bool;
            GluingFault : Bool;
            GluingRefillTank : Bool;
            GluingTankEmpty : Bool;
            "8" : Bool;
            "9" : Bool;
            "10" : Bool;
            "11" : Bool;
            "12" : Bool;
            "13" : Bool;
            "14" : Bool;
            "15" : Bool;
            "16" : Bool;
         END_STRUCT;
         C_Spare_3 : Struct
            "1" : Bool;
            "2" : Bool;
            "3" : Bool;
            "4" : Bool;
            "5" : Bool;
            "6" : Bool;
            "7" : Bool;
            "8" : Bool;
            "9" : Bool;
            "10" : Bool;
            "11" : Bool;
            "12" : Bool;
            "13" : Bool;
            "14" : Bool;
            "15" : Bool;
            "16" : Bool;
         END_STRUCT;
         C_Spare_4 : Struct
            "1" : Bool;
            "2" : Bool;
            "3" : Bool;
            "4" : Bool;
            "5" : Bool;
            "6" : Bool;
            "7" : Bool;
            "8" : Bool;
            "9" : Bool;
            "10" : Bool;
            "11" : Bool;
            "12" : Bool;
            "13" : Bool;
            "14" : Bool;
            "15" : Bool;
            "16" : Bool;
         END_STRUCT;
      END_STRUCT;
      "E" : Struct   // 上料扫码错误
         NG_1 : Struct
            ShaftScanNGFull : Bool;
            PressNGFull : Bool;
            RingScanNGFull : Bool;
            ShaftScanStatus : Bool;
            PressNGStatus : Bool;
            RingScanNGStatus : Bool;
            "NG 1 DoorOpen" : Bool;
            "NG 2 DoorOpen" : Bool;
            "9" : Bool;
            "10" : Bool;
            "11" : Bool;
            "12" : Bool;
            "13" : Bool;
            "14" : Bool;
            "15" : Bool;
            "16" : Bool;
         END_STRUCT;
         NG_2 : Struct
            "Press/GlueNGFull" : Bool;
            MagnetNGFull : Bool;
            RingScanNGFull : Bool;
            "Press/GlueNGStatus" : Bool;
            MagnetNGStatus : Bool;
            RingScanNGStatus : Bool;
            "7" : Bool;
            "8" : Bool;
            "9" : Bool;
            "10" : Bool;
            "11" : Bool;
            "12" : Bool;
            "13" : Bool;
            "14" : Bool;
            "15" : Bool;
            "16" : Bool;
         END_STRUCT;
         E_Spare_1 : Struct
            "1" : Bool;
            "2" : Bool;
            "3" : Bool;
            "4" : Bool;
            "5" : Bool;
            "6" : Bool;
            "7" : Bool;
            "8" : Bool;
            "9" : Bool;
            "10" : Bool;
            "11" : Bool;
            "12" : Bool;
            "13" : Bool;
            "14" : Bool;
            "15" : Bool;
            "16" : Bool;
         END_STRUCT;
         E_Spare_2 : Struct
            "1" : Bool;
            "2" : Bool;
            "3" : Bool;
            "4" : Bool;
            "5" : Bool;
            "6" : Bool;
            "7" : Bool;
            "8" : Bool;
            "9" : Bool;
            "10" : Bool;
            "11" : Bool;
            "12" : Bool;
            "13" : Bool;
            "14" : Bool;
            "15" : Bool;
            "16" : Bool;
         END_STRUCT;
         E_Spare_3 : Struct
            "1" : Bool;
            "2" : Bool;
            "3" : Bool;
            "4" : Bool;
            "5" : Bool;
            "6" : Bool;
            "7" : Bool;
            "8" : Bool;
            "9" : Bool;
            "10" : Bool;
            "11" : Bool;
            "12" : Bool;
            "13" : Bool;
            "14" : Bool;
            "15" : Bool;
            "16" : Bool;
         END_STRUCT;
      END_STRUCT;
      F : Struct   // RFID错误
         Robot_1 : Struct
            Grip1Error : Bool;
            Grip2Error : Bool;
            Grip1SensorCheckError : Bool;
            Grip2SensorCheckError : Bool;
            ManualMoved : Bool;
            "EXT Fault" : Bool;
            RobotNOTStart : Bool;
            "8" : Bool;
            "9" : Bool;
            "10" : Bool;
            "11" : Bool;
            "12" : Bool;
            "13" : Bool;
            "14" : Bool;
            "15" : Bool;
            "16" : Bool;
         END_STRUCT;
         Robot_2 : Struct
            Grip1Error : Bool;
            Grip2Error : Bool;
            Grip1SensorCheckError : Bool;
            Grip2SensorCheckError : Bool;
            ManualMoved : Bool;
            ReadNG_1 : Bool;
            ReadNG_2 : Bool;
            ReadNG_3 : Bool;
            ReadNG_4 : Bool;
            "EXT Fault" : Bool;
            RobotNOTStart : Bool;
            "12" : Bool;
            "13" : Bool;
            "14" : Bool;
            "15" : Bool;
            "16" : Bool;
         END_STRUCT;
         Robot_3 : Struct
            Grip1Error : Bool;
            Grip2Error : Bool;
            Grip1SensorCheckError : Bool;
            Grip2SensorCheckError : Bool;
            ManualMoved : Bool;
            "EXT Fault" : Bool;
            RobotNOTStart : Bool;
            "8" : Bool;
            "9" : Bool;
            "10" : Bool;
            "11" : Bool;
            "12" : Bool;
            "13" : Bool;
            "14" : Bool;
            "15" : Bool;
            "16" : Bool;
         END_STRUCT;
         F_Spare_1 : Struct
            Scan_805A1 : Bool;
            Robot_1 : Bool;
            Robot_2 : Bool;
            Robot_3 : Bool;
            "5" : Bool;
            "6" : Bool;
            "7" : Bool;
            "8" : Bool;
            "9" : Bool;
            "10" : Bool;
            "11" : Bool;
            "12" : Bool;
            "13" : Bool;
            "14" : Bool;
            "15" : Bool;
            "16" : Bool;
         END_STRUCT;
         F_Spare_2 : Struct
            "1" : Bool;
            "2" : Bool;
            "3" : Bool;
            "4" : Bool;
            "5" : Bool;
            "6" : Bool;
            "7" : Bool;
            "8" : Bool;
            "9" : Bool;
            "10" : Bool;
            "11" : Bool;
            "12" : Bool;
            "13" : Bool;
            "14" : Bool;
            "15" : Bool;
            "16" : Bool;
         END_STRUCT;
      END_STRUCT;
      H : Struct   // B-打标模组激光打标机1错误
         ShaftLine : Struct   // Total Error Status, Use for error code
            LiftingCylStatusError : Bool;
            LoadingStop1timeout : Bool;
            LoadingStop2timeout : Bool;
            LoadingStop3timeout : Bool;
            LoadingStop4timeout : Bool;
            UnloadingStop1timeout : Bool;
            UnloadingStop2timeout : Bool;
            UnloadingStop3timeout : Bool;
            UnloadingLiftingtimeout : Bool;
            EmptyStop1timeout : Bool;
            EmptyStop2timeout : Bool;
            EmptyStop3timeout : Bool;
            EmptyStop4timeout : Bool;
            "14" : Bool;
            "15" : Bool;
            "16" : Bool;
         END_STRUCT;
         Spare_1 : Struct
            "H-shaftLifting_Motor" : Bool;
            "H-shaftLoad_Motor" : Bool;
            "H-shaftUnLoad_Motor" : Bool;
            "4" : Bool;
            "5" : Bool;
            "6" : Bool;
            "7" : Bool;
            "8" : Bool;
            "9" : Bool;
            "10" : Bool;
            "11" : Bool;
            "12" : Bool;
            "13" : Bool;
            "14" : Bool;
            "15" : Bool;
            "16" : Bool;
         END_STRUCT;
         Spare_2 : Struct
            "1" : Bool;
            "2" : Bool;
            "3" : Bool;
            "4" : Bool;
            "5" : Bool;
            "6" : Bool;
            "7" : Bool;
            "8" : Bool;
            "9" : Bool;
            "10" : Bool;
            "11" : Bool;
            "12" : Bool;
            "13" : Bool;
            "14" : Bool;
            "15" : Bool;
            "16" : Bool;
         END_STRUCT;
         Spare_3 : Struct
            "1" : Bool;
            "2" : Bool;
            "3" : Bool;
            "4" : Bool;
            "5" : Bool;
            "6" : Bool;
            "7" : Bool;
            "8" : Bool;
            "9" : Bool;
            "10" : Bool;
            "11" : Bool;
            "12" : Bool;
            "13" : Bool;
            "14" : Bool;
            "15" : Bool;
            "16" : Bool;
         END_STRUCT;
         Spare_4 : Struct
            "1" : Bool;
            "2" : Bool;
            "3" : Bool;
            "4" : Bool;
            "5" : Bool;
            "6" : Bool;
            "7" : Bool;
            "8" : Bool;
            "9" : Bool;
            "10" : Bool;
            "11" : Bool;
            "12" : Bool;
            "13" : Bool;
            "14" : Bool;
            "15" : Bool;
            "16" : Bool;
         END_STRUCT;
      END_STRUCT;
      J : Struct
         MagnetLine : Struct   // Total Error Status, Use for error code
            LiftingCylStatusError : Bool;
            LoadingStop1timeout : Bool;
            LoadingStop2timeout : Bool;
            LoadingStop3timeout : Bool;
            LoadingStop4timeout : Bool;
            UnloadingStop1timeout : Bool;
            UnloadingStop2timeout : Bool;
            UnloadingStop3timeout : Bool;
            UnloadingLiftingtimeout : Bool;
            EmptyStop1timeout : Bool;
            EmptyStop2timeout : Bool;
            EmptyStop3timeout : Bool;
            EmptyStop4timeout : Bool;
            "14" : Bool;
            "15" : Bool;
            "16" : Bool;
         END_STRUCT;
         Spare_1 : Struct
            "J-MagnetLifting_Motor" : Bool;
            "J-MagnetLoad_Motor" : Bool;
            "J-MagnetUnLoad_Motor" : Bool;
            "4" : Bool;
            "5" : Bool;
            "6" : Bool;
            "7" : Bool;
            "8" : Bool;
            "9" : Bool;
            "10" : Bool;
            "11" : Bool;
            "12" : Bool;
            "13" : Bool;
            "14" : Bool;
            "15" : Bool;
            "16" : Bool;
         END_STRUCT;
         Spare_2 : Struct
            "1" : Bool;
            "2" : Bool;
            "3" : Bool;
            "4" : Bool;
            "5" : Bool;
            "6" : Bool;
            "7" : Bool;
            "8" : Bool;
            "9" : Bool;
            "10" : Bool;
            "11" : Bool;
            "12" : Bool;
            "13" : Bool;
            "14" : Bool;
            "15" : Bool;
            "16" : Bool;
         END_STRUCT;
         Spare_3 : Struct
            "1" : Bool;
            "2" : Bool;
            "3" : Bool;
            "4" : Bool;
            "5" : Bool;
            "6" : Bool;
            "7" : Bool;
            "8" : Bool;
            "9" : Bool;
            "10" : Bool;
            "11" : Bool;
            "12" : Bool;
            "13" : Bool;
            "14" : Bool;
            "15" : Bool;
            "16" : Bool;
         END_STRUCT;
         Spare_4 : Struct
            "1" : Bool;
            "2" : Bool;
            "3" : Bool;
            "4" : Bool;
            "5" : Bool;
            "6" : Bool;
            "7" : Bool;
            "8" : Bool;
            "9" : Bool;
            "10" : Bool;
            "11" : Bool;
            "12" : Bool;
            "13" : Bool;
            "14" : Bool;
            "15" : Bool;
            "16" : Bool;
         END_STRUCT;
      END_STRUCT;
      K : Struct
         ReserveLine : Struct   // Total Error Status, Use for error code
            LiftingCylStatusError : Bool;
            LoadingStop1timeout : Bool;
            LoadingStop2timeout : Bool;
            LoadingStop3timeout : Bool;
            LoadingStop4timeout : Bool;
            UnloadingStop1timeout : Bool;
            UnloadingStop2timeout : Bool;
            UnloadingStop3timeout : Bool;
            UnloadingLiftingtimeout : Bool;
            EmptyStop1timeout : Bool;
            EmptyStop2timeout : Bool;
            EmptyStop3timeout : Bool;
            EmptyStop4timeout : Bool;
            "14" : Bool;
            "15" : Bool;
            "16" : Bool;
         END_STRUCT;
         Spare_1 : Struct
            "K-Lifting_Motor" : Bool;
            "K-ReserveLoad_Motor" : Bool;
            "K-ReserveUnLoad_Motor" : Bool;
            "4" : Bool;
            "5" : Bool;
            "6" : Bool;
            "7" : Bool;
            "8" : Bool;
            "9" : Bool;
            "10" : Bool;
            "11" : Bool;
            "12" : Bool;
            "13" : Bool;
            "14" : Bool;
            "15" : Bool;
            "16" : Bool;
         END_STRUCT;
         Spare_2 : Struct
            "1" : Bool;
            "2" : Bool;
            "3" : Bool;
            "4" : Bool;
            "5" : Bool;
            "6" : Bool;
            "7" : Bool;
            "8" : Bool;
            "9" : Bool;
            "10" : Bool;
            "11" : Bool;
            "12" : Bool;
            "13" : Bool;
            "14" : Bool;
            "15" : Bool;
            "16" : Bool;
         END_STRUCT;
         Spare_3 : Struct
            "1" : Bool;
            "2" : Bool;
            "3" : Bool;
            "4" : Bool;
            "5" : Bool;
            "6" : Bool;
            "7" : Bool;
            "8" : Bool;
            "9" : Bool;
            "10" : Bool;
            "11" : Bool;
            "12" : Bool;
            "13" : Bool;
            "14" : Bool;
            "15" : Bool;
            "16" : Bool;
         END_STRUCT;
         Spare_4 : Struct
            "1" : Bool;
            "2" : Bool;
            "3" : Bool;
            "4" : Bool;
            "5" : Bool;
            "6" : Bool;
            "7" : Bool;
            "8" : Bool;
            "9" : Bool;
            "10" : Bool;
            "11" : Bool;
            "12" : Bool;
            "13" : Bool;
            "14" : Bool;
            "15" : Bool;
            "16" : Bool;
         END_STRUCT;
      END_STRUCT;
      L : Struct
         UnloadingLine : Struct   // Total Error Status, Use for error code
            UnloadingTransCylinderError : Bool;
            LoadingStop1timeout : Bool;
            LoadingStop2timeout : Bool;
            LoadingStop3timeout : Bool;
            LoadingStop4timeout : Bool;
            UnloadingStop1timeout : Bool;
            UnloadingStop2timeout : Bool;
            UnloadingStop3timeout : Bool;
            UnloadingLiftingtimeout : Bool;
            EmptyStop1timeout : Bool;
            EmptyStop2timeout : Bool;
            EmptyStop3timeout : Bool;
            EmptyStop4timeout : Bool;
            "14" : Bool;
            "15" : Bool;
            "16" : Bool;
         END_STRUCT;
         CuringOven : Struct
            "1" : Bool;
            "2" : Bool;
            "3" : Bool;
            "4" : Bool;
            "5" : Bool;
            "6" : Bool;
            "7" : Bool;
            "8" : Bool;
            "9" : Bool;
            "10" : Bool;
            "11" : Bool;
            "12" : Bool;
            "13" : Bool;
            "14" : Bool;
            "15" : Bool;
            "16" : Bool;
         END_STRUCT;
         Spare_2 : Struct
            "L-Unloading_Motor" : Bool;
            "L-Unloading _LineMotor" : Bool;
            "3" : Bool;
            "4" : Bool;
            "5" : Bool;
            "6" : Bool;
            "7" : Bool;
            "8" : Bool;
            "9" : Bool;
            "10" : Bool;
            "11" : Bool;
            "12" : Bool;
            "13" : Bool;
            "14" : Bool;
            "15" : Bool;
            "16" : Bool;
         END_STRUCT;
         Spare_3 : Struct
            "1" : Bool;
            "2" : Bool;
            "3" : Bool;
            "4" : Bool;
            "5" : Bool;
            "6" : Bool;
            "7" : Bool;
            "8" : Bool;
            "9" : Bool;
            "10" : Bool;
            "11" : Bool;
            "12" : Bool;
            "13" : Bool;
            "14" : Bool;
            "15" : Bool;
            "16" : Bool;
         END_STRUCT;
         Spare_4 : Struct
            "1" : Bool;
            "2" : Bool;
            "3" : Bool;
            "4" : Bool;
            "5" : Bool;
            "6" : Bool;
            "7" : Bool;
            "8" : Bool;
            "9" : Bool;
            "10" : Bool;
            "11" : Bool;
            "12" : Bool;
            "13" : Bool;
            "14" : Bool;
            "15" : Bool;
            "16" : Bool;
         END_STRUCT;
      END_STRUCT;
      MES_Error : Struct
         Offline : Bool;   // MES离线
         Reserved1_8 : Bool;
         CheckInCompOverTime_1 : Bool;   // 心跳故障
         CheckInResultOverTime_1 : Bool;
         CheckInCompOverTime_2 : Bool;   // 二维码对比失败
         CheckInResultOverTime_2 : Bool;   // 获取打标数据NG
         CheckInCompOverTime_3 : Bool;   // 获取打标数据超时
         CheckInResultOverTime_3 : Bool;   // 缓存数据和MES数据对比不合格，步序错误 需初始化
         CheckInCompOverTime_4 : Bool;
         CheckInResultOverTime_4 : Bool;   // 主件查询完成超时
         CheckInCompOverTime_5 : Bool;   // 主件查询结果NG
         CheckInResultOverTime_5 : Bool;   // 主件查询完成复位超时
         CheckInCompOverTime_6 : Bool;
         CheckInResultOverTime_6 : Bool;
         CheckInCompOverTime_7 : Bool;
         CheckInResultOverTime_7 : Bool;   // 主件保存完成超时
         CheckInCompOverTime_8 : Bool;   // 主件保存结果反馈超时
         CheckInResultOverTime_8 : Bool;   // 主件保存触发错误
         CheckoutSaveResultNG : Bool;   // 主件保存结果NG
         CheckoutCompRstOverTime : Bool;   // 主件保存完成复位超时
         Reserved2_5 : Bool;
         Reserved2_6 : Bool;
         Reserved2_7 : Bool;
         SubCheck_CompOverTime : Bool;   // 子件查询完成超时
         SubCheck_ResultOverTime : Bool;   // 子件查询结果反馈超时
         SubCheck_TriggerError : Bool;   // 子件查询触发错误
         SubCheck_CheckResultNG : Bool;   // 子件查询结果NG
         SubCheck_CompRstOverTime : Bool;   // 子件查询完成复位超时
         Reserved3_5 : Bool;
         Reserved3_6 : Bool;
         Reserved3_7 : Bool;
         Processing_CompOverTime : Bool;   // 加工不可逆标记完成超时
         Reserved4_1 : Bool;
         Processing_TriggerError : Bool;   // 加工不可逆标记触发错误
         Reserved4_3 : Bool;
         Processing_CompRstOverTime : Bool;   // 加工不可逆标记完成复位超时
         Reserved4_5 : Bool;
         Reserved4_6 : Bool;
         Reserved4_7 : Bool;
         Reserved5_0 : Bool;
         Reserved5_1 : Bool;
         Reserved5_2 : Bool;
         Reserved5_3 : Bool;
         Reserved5_4 : Bool;
         Reserved5_5 : Bool;
         Reserved5_6 : Bool;
         Reserved5_7 : Bool;
      END_STRUCT;
   END_VAR
BEGIN
END_DATA_BLOCK
